ABB RobotStudio station: Tp2_20201212-055033.rsstn

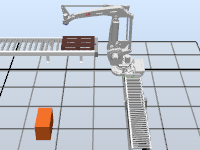
Station Tp2 (saved by RobotStudio 20.1.8982.0)
Layout (positions relative to the parent item):
  - IRB660_180_315__01 [mechanism, from Robots\IRB660_180_315__01.rslib] at (0, 0, 0) mm; joint values [0.0199, 0, 0, 0] (rad or m)
  - transporteCajas [part, from Equipment\Conveyor Guide 400.rslib] at (0, 1500, 0) mm, rotated rx 0 ry 0 rz 90 deg
  - Euro Pallet [graphiccomponentgroup, from Equipment\Euro Pallet.rslib] at (1000, -1425, 435) mm
    - Body 1 [part, from Equipment\Euro Pallet.rslib]
  - transportePallets [part, from Equipment\Conveyor 950 4000 h2.rslib] at (1000, -1500, 0) mm
  - caja [part] at (2366.26, 2652.95, 0) mm
  - topePallet [frame] at (1000, -1025, 435) mm
  - basePallet [frame] at (1000, -1025, 435) mm
  - topeCajas [frame] at (-200, 1500, 770) mm
Attachment: Euro Pallet is attached to transportePallets
Attachment: basePallet is attached to Euro Pallet
Attachment: topePallet is attached to transportePallets
Attachment: topeCajas is attached to transporteCajas
